TYPE MDP5001_341_I_7CD731EE :
STRUCT
	MDP5001_341_L1_Status_Voltage_Sign_Bit			: BIT;
	MDP5001_341_L1_Status_Overvoltage				: BIT;
	MDP5001_341_L1_Status_Overcurrent				: BIT;
	MDP5001_341_L1_Status_Inaccurate_Voltage		: BIT;
	MDP5001_341_L1_Status_Inaccurate_Current		: BIT;
	MDP5001_341_L1_Status_Voltage_Guard_Warning		: BIT;
	MDP5001_341_L1_Status_Voltage_Guard_Error		: BIT;
	MDP5001_341_L1_Status_Current_Guard_Warning		: BIT;
	MDP5001_341_L1_Status_Current_Guard_Error		: BIT;
	MDP5001_341_L1_Status_TxPDO_Toggle				: BIT;
	MDP5001_341_L1_Basic_Voltage					: REAL;
	MDP5001_341_L1_Basic_Current					: REAL;
	MDP5001_341_L1_Power_Active_Power				: REAL;
	MDP5001_341_L1_Power_Apparent_Power				: REAL;
	MDP5001_341_L1_Power_Reactive_Power				: REAL;
	MDP5001_341_L1_Power_Power_Factor				: REAL;
	MDP5001_341_L2_Status_Voltage_Sign_Bit			: BIT;
	MDP5001_341_L2_Status_Overvoltage				: BIT;
	MDP5001_341_L2_Status_Overcurrent				: BIT;
	MDP5001_341_L2_Status_Inaccurate_Voltage		: BIT;
	MDP5001_341_L2_Status_Inaccurate_Current		: BIT;
	MDP5001_341_L2_Status_Voltage_Guard_Warning		: BIT;
	MDP5001_341_L2_Status_Voltage_Guard_Error		: BIT;
	MDP5001_341_L2_Status_Current_Guard_Warning		: BIT;
	MDP5001_341_L2_Status_Current_Guard_Error		: BIT;
	MDP5001_341_L2_Status_TxPDO_Toggle				: BIT;
	MDP5001_341_L2_Basic_Voltage					: REAL;
	MDP5001_341_L2_Basic_Current					: REAL;
	MDP5001_341_L2_Power_Active_Power				: REAL;
	MDP5001_341_L2_Power_Apparent_Power				: REAL;
	MDP5001_341_L2_Power_Reactive_Power				: REAL;
	MDP5001_341_L2_Power_Power_Factor				: REAL;
	MDP5001_341_L3_Status_Voltage_Sign_Bit			: BIT;
	MDP5001_341_L3_Status_Overvoltage				: BIT;
	MDP5001_341_L3_Status_Overcurrent				: BIT;
	MDP5001_341_L3_Status_Inaccurate_Voltage		: BIT;
	MDP5001_341_L3_Status_Inaccurate_Current		: BIT;
	MDP5001_341_L3_Status_Voltage_Guard_Warning		: BIT;
	MDP5001_341_L3_Status_Voltage_Guard_Error		: BIT;
	MDP5001_341_L3_Status_Current_Guard_Warning		: BIT;
	MDP5001_341_L3_Status_Current_Guard_Error		: BIT;
	MDP5001_341_L3_Status_TxPDO_Toggle				: BIT;
	MDP5001_341_L3_Basic_Voltage					: REAL;
	MDP5001_341_L3_Basic_Current					: REAL;
	MDP5001_341_L3_Power_Active_Power				: REAL;
	MDP5001_341_L3_Power_Apparent_Power				: REAL;
	MDP5001_341_L3_Power_Reactive_Power				: REAL;
	MDP5001_341_L3_Power_Power_Factor				: REAL;	
	MDP5001_341_Total_Status_System_State					: BIT;
	MDP5001_341_Total_Status_Grid_Direction					: BIT;
	MDP5001_341_Total_Status_Frequency_Guard_Warning		: BIT;
	MDP5001_341_Total_Status_Frequency_Guard_Error			: BIT;
	MDP5001_341_Total_Status_Neutral_Current_Guard_Warning	: BIT;
	MDP5001_341_Total_Status_Neutral_Current_Guard_Error	: BIT;
	MDP5001_341_Total_Status_Active_Power_Guard_Warning		: BIT;
	MDP5001_341_Total_Status_Active_Power_Guard_Error		: BIT;
	MDP5001_341_Total_Status_Apparent_Power_Guard_Warning	: BIT;
	MDP5001_341_Total_Status_Apparent_Power_Guard_Error		: BIT;
	MDP5001_341_Total_Status_Power_Quality_Guard_Warning	: BIT;
	MDP5001_341_Total_Status_Power_Quality_Guard_Error		: BIT;
	MDP5001_341_Total_Status_TxPDO_State					: BIT;
	MDP5001_341_Total_Status_TxPDO_Toggle					: BIT;
	MDP5001_341_Total_Status_Power_Quality_Factor			: REAL;	
	MDP5001_341_Total_Basic_Frequency						: REAL;	
	MDP5001_341_Total_Basic_Power_Factor					: REAL;	
	MDP5001_341_Total_Basic_Calculated_Neutral_Line_Current	: REAL;	
	MDP5001_341_Total_Variant_Value_In_TxPDO_Toggle			: BIT;
	MDP5001_341_Total_Variant_Value_In_Index_1_REAL			: UINT;
	MDP5001_341_Total_Variant_Value_In_Value_1_REAL			: REAL;
	MDP5001_341_Total_Variant_Value_In_Index_2_REAL			: UINT;
	MDP5001_341_Total_Variant_Value_In_Value_2_REAL			: REAL;
	MDP5001_341_Total_Variant_Value_In_Index_3_REAL			: UINT;
	MDP5001_341_Total_Variant_Value_In_Value_3_REAL			: REAL;
	MDP5001_341_Total_Variant_Value_In_Index_4_ULINT		: UINT;
	MDP5001_341_Total_Variant_Value_In_Value_4_ULINT		: ULINT;
	MDP5001_341_DPM_Data_Data_1								: UDINT;
	MDP5001_341_DPM_Data_Data_2								: UDINT;
	MDP5001_341_DPM_Data_Data_3								: UDINT;
	MDP5001_341_DPM_Data_Data_4								: UDINT;
	MDP5001_341_DPM_Data_Data_5								: UDINT;
	MDP5001_341_DPM_Data_Data_6								: UDINT;
	MDP5001_341_DPM_Data_Data_7								: UDINT;
	MDP5001_341_DPM_Data_Data_8								: UDINT;
	MDP5001_341_DPM_Data_Data_9								: UDINT;
	MDP5001_341_DPM_Data_Data_10							: UDINT;
	MDP5001_341_DPM_Data_Data_11							: UDINT;
	MDP5001_341_DPM_Data_Data_12							: UDINT;
	MDP5001_341_DPM_Data_Data_13							: UDINT;
	MDP5001_341_DPM_Data_Data_14							: UDINT;
	MDP5001_341_DPM_Data_Data_15							: UDINT;
	MDP5001_341_DPM_Data_Data_16							: UDINT;
	MDP5001_341_DPM_Data_Data_17							: UDINT;
	MDP5001_341_DPM_Data_Data_18							: UDINT;
	MDP5001_341_DPM_Data_Data_19							: UDINT;
	MDP5001_341_DPM_Data_Data_20							: UDINT;
END_STRUCT
END_TYPE

(* stored: Version 1.1.0.1, ProductVersion 3.1.4024.12
   DUT MDP5001_341_I_7CD731EE: Id {895cf906-2b33-49e9-9919-d5e363b63523} *)
